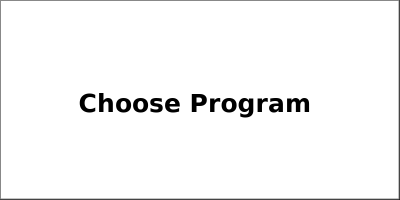
VISUALIZATION V_ProductionWelcome  // 400x200
    RoundedRectangle (0,0 400x200)
    Label (41,53 308x100), "Choose Program"
END_VISUALIZATION

(* stored: Version 1.1.0.1, ProductVersion 3.1.4024.15
   Visu V_ProductionWelcome: Id {b3fd8b1a-71ef-461a-9087-d3a02270569f} *)
